PROGRAM Test_FilePOU
VAR
	testMetho:FB_FileGets;
END_VAR

testMetho(
	sNetId:= , 
	hFile:= , 
	bExecute:= , 
	tTimeout:= , 
	bBusy=> , 
	bError=> , 
	nErrId=> , 
	sLine=> , 
	bEOF=> );

END_PROGRAM

(* stored: Version 1.1.0.1, ProductVersion 3.1.4024.4
   POU Test_FilePOU: Id {76bd06bd-c875-45f8-8e4a-dba25291c55d}, SpecialFunc None *)
